// TIA Portal project "selector" (V16)

(* hardware
DEVICE "S7-1200 station_1"  S7-1200 Station
   slot 0: "Rack_0"  S7-1200 Rack  Rack  V1.0
   slot 1: "PLC_1"  CPU 1212C AC/DC/Rly  6ES7 212-1BE40-0XB0  V4.0
*)

// ===== PLC "PLC_1"  CPU 1212C AC/DC/Rly =====

VAR_GLOBAL   // PLC tag table "Default tag table"
   "selector 1" AT %I0.0 : Bool;
   "selector 2" AT %I0.1 : Bool;
   "km1" AT %Q0.0 : Bool;
   "km2" AT %Q0.1 : Bool;
   "km3" AT %Q0.2 : Bool;
   "Tag_1" AT %M0.0 : Bool;
   "Tag_2" AT %M0.1 : Bool;
   "Tag_3" AT %M0.2 : Bool;
   "Tag_4" AT %M0.3 : Bool;
   "Tag_5" AT %M0.5 : Bool;
   "Tag_6" AT %M0.4 : Bool;
   "Tag_7" AT %M1.0 : Bool;
END_VAR

// folder: System blocks/Program resources

DATA_BLOCK "T1-1"   // DB1
{ S7_Optimized_Access := 'TRUE' }
AUTHOR : Simatic
FAMILY : IEC
NAME : IEC_TMR
VERSION : 1.0
// stored: InstanceOfName IEC_TIMER
"IEC_TIMER"
BEGIN
END_DATA_BLOCK

DATA_BLOCK "T1-2"   // DB2
{ S7_Optimized_Access := 'TRUE' }
AUTHOR : Simatic
FAMILY : IEC
NAME : IEC_TMR
VERSION : 1.0
// stored: InstanceOfName IEC_TIMER
"IEC_TIMER"
BEGIN
END_DATA_BLOCK

DATA_BLOCK "T2-1"   // DB3
{ S7_Optimized_Access := 'TRUE' }
AUTHOR : Simatic
FAMILY : IEC
NAME : IEC_TMR
VERSION : 1.0
// stored: InstanceOfName IEC_TIMER
"IEC_TIMER"
BEGIN
END_DATA_BLOCK

DATA_BLOCK "T2-2"   // DB4
{ S7_Optimized_Access := 'TRUE' }
AUTHOR : Simatic
FAMILY : IEC
NAME : IEC_TMR
VERSION : 1.0
// stored: InstanceOfName IEC_TIMER
"IEC_TIMER"
BEGIN
END_DATA_BLOCK

DATA_BLOCK "T2-3"   // DB5
{ S7_Optimized_Access := 'TRUE' }
AUTHOR : Simatic
FAMILY : IEC
NAME : IEC_TMR
VERSION : 1.0
// stored: InstanceOfName IEC_TIMER
"IEC_TIMER"
BEGIN
END_DATA_BLOCK

// folder: (top level)

ORGANIZATION_BLOCK "Main"   // OB1, LAD, ProgramCycle
TITLE = "Main Program Sweep (Cycle)"
{ S7_Optimized_Access := 'TRUE' }
VERSION : 0.1
   VAR_INPUT
      Initial_Call : Bool;   // Initial call of this OB
      Remanence : Bool;   // =True, if remanent data are available
   END_VAR
   VAR_TEMP   // added for the SCL form of the ladder/FBD networks
      _w1 : Bool;
   END_VAR
BEGIN

REGION Network 1
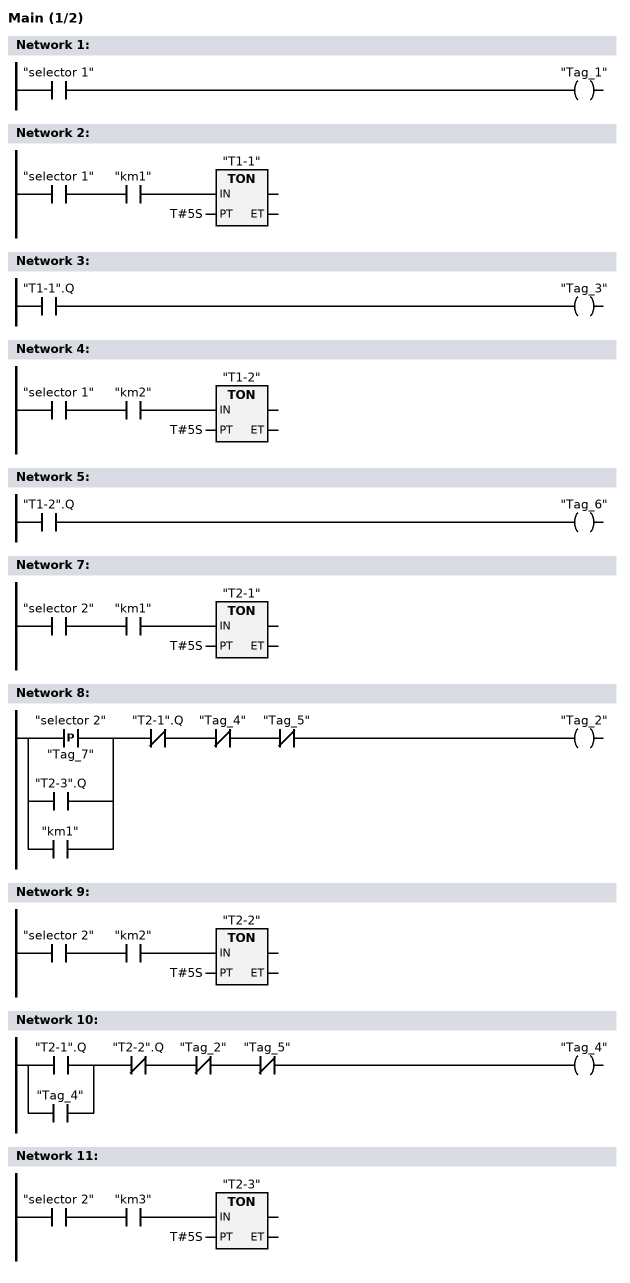
   RUNG wire#powerrail
      Contact( "selector 1" )
      Coil( "Tag_1" )
   END_RUNG
   // the same network as SCL:
   "Tag_1" := "selector 1";
END_REGION

REGION Network 2
   "T1-1".TON(IN := "selector 1" AND "km1", PT := T#5S);
END_REGION

REGION Network 3
   RUNG wire#powerrail
      Contact( "T1-1".Q )
      Coil( "Tag_3" )
   END_RUNG
   // the same network as SCL:
   "Tag_3" := "T1-1".Q;
END_REGION

REGION Network 4
   "T1-2".TON(IN := "selector 1" AND "km2", PT := T#5S);
END_REGION

REGION Network 5
   RUNG wire#powerrail
      Contact( "T1-2".Q )
      Coil( "Tag_6" )
   END_RUNG
   // the same network as SCL:
   "Tag_6" := "T1-2".Q;
END_REGION

REGION Network 7
   "T2-1".TON(IN := "selector 2" AND "km1", PT := T#5S);
END_REGION

REGION Network 8
   RUNG wire#powerrail
      P_Contact(operand := "selector 2", bit := "Tag_7")
      wire#w1
      I_Contact( "T2-1".Q )
      I_Contact( "Tag_4" )
      I_Contact( "Tag_5" )
      Coil( "Tag_2" )
   END_RUNG
   RUNG wire#powerrail
      Contact( "T2-3".Q )
   END_RUNG wire#w1
   RUNG wire#powerrail
      Contact( "km1" )
   END_RUNG wire#w1
   // the same network as SCL:
   #_w1 := "selector 2" AND NOT "Tag_7";   // rising edge of "selector 2"
   "Tag_7" := "selector 2";
   "Tag_2" := (#_w1 OR "T2-3".Q OR "km1") AND NOT "T2-1".Q AND NOT "Tag_4" AND NOT "Tag_5";
END_REGION

REGION Network 9
   "T2-2".TON(IN := "selector 2" AND "km2", PT := T#5S);
END_REGION

REGION Network 10
   RUNG wire#powerrail
      Contact( "T2-1".Q )
      wire#w1
      I_Contact( "T2-2".Q )
      I_Contact( "Tag_2" )
      I_Contact( "Tag_5" )
      Coil( "Tag_4" )
   END_RUNG
   RUNG wire#powerrail
      Contact( "Tag_4" )
   END_RUNG wire#w1
   // the same network as SCL:
   "Tag_4" := ("T2-1".Q OR "Tag_4") AND NOT "T2-2".Q AND NOT "Tag_2" AND NOT "Tag_5";
END_REGION

REGION Network 11
   "T2-3".TON(IN := "selector 2" AND "km3", PT := T#5S);
END_REGION

REGION Network 12
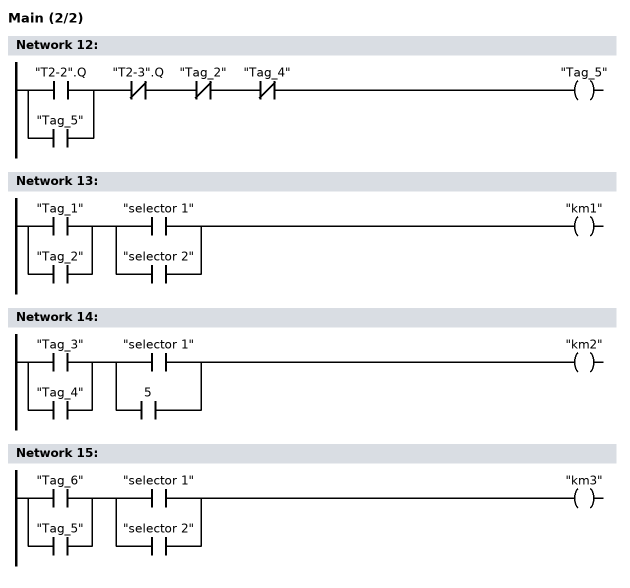
   RUNG wire#powerrail
      Contact( "T2-2".Q )
      wire#w1
      I_Contact( "T2-3".Q )
      I_Contact( "Tag_2" )
      I_Contact( "Tag_4" )
      Coil( "Tag_5" )
   END_RUNG
   RUNG wire#powerrail
      Contact( "Tag_5" )
   END_RUNG wire#w1
   // the same network as SCL:
   "Tag_5" := ("T2-2".Q OR "Tag_5") AND NOT "T2-3".Q AND NOT "Tag_2" AND NOT "Tag_4";
END_REGION

REGION Network 13
   RUNG wire#powerrail
      Contact( "Tag_1" )
      wire#w1
      Contact( "selector 1" )
      wire#w2
      Coil( "km1" )
   END_RUNG
   RUNG wire#powerrail
      Contact( "Tag_2" )
   END_RUNG wire#w1
   RUNG wire#w1
      Contact( "selector 2" )
   END_RUNG wire#w2
   // the same network as SCL:
   "km1" := ("Tag_1" OR "Tag_2") AND ("selector 1" OR "selector 2");
END_REGION

REGION Network 14
   RUNG wire#powerrail
      Contact( "Tag_3" )
      wire#w1
      Contact( "selector 1" )
      wire#w2
      Coil( "km2" )
   END_RUNG
   RUNG wire#powerrail
      Contact( "Tag_4" )
   END_RUNG wire#w1
   RUNG wire#w1
      Contact( 5 )
   END_RUNG wire#w2
   // the same network as SCL:
   "km2" := ("Tag_3" OR "Tag_4") AND ("selector 1" OR 5);
END_REGION

REGION Network 15
   RUNG wire#powerrail
      Contact( "Tag_6" )
      wire#w1
      Contact( "selector 1" )
      wire#w2
      Coil( "km3" )
   END_RUNG
   RUNG wire#powerrail
      Contact( "Tag_5" )
   END_RUNG wire#w1
   RUNG wire#w1
      Contact( "selector 2" )
   END_RUNG wire#w2
   // the same network as SCL:
   "km3" := ("Tag_6" OR "Tag_5") AND ("selector 1" OR "selector 2");
END_REGION
END_ORGANIZATION_BLOCK